Staubli VAL3: MoveToPoint.pgx

program MoveToPoint()
  local num l_nStatus
  local num l_nWorkMode
  local num l_ni
begin
  //
  link(pTemp,fFrmTemp)
  while true
    l_nWorkMode=workingMode(l_nStatus)
    if l_nWorkMode==1 and l_nStatus==0
      pTemp.trsf=pdemo[nSelected].trsf
      pTemp.config=pdemo[nSelected].config
      movel(pTemp,t2,mSuDu[1])
    else
      resetMotion()
    endIf
  endWhile
  //
end
